PROGRAM MAIN
VAR
	// ------ Linking variables to IO cards ------
		// --------- Outputs ---------
	Flow_Valve_1 	AT %Q* : INT;
	Level_Valve_1 	AT %Q* : INT;
	Level_Valve_2 	AT %Q* : INT;
	Level_Valve_3 	AT %Q* : INT;
	Gas_Valve 		AT %Q* : INT;
	Mixer_Valve 	AT %Q* : INT;
	Motor_speed 	AT %Q* : INT;	
	Motor_Direction AT %Q* : BOOL; 			// Don't touch
		// --------- Inputs ---------
			// Buttons
	Toggle_Button 	AT %I* :BOOL;	// Normally Open  (OFF), Green
	Reset_Button 	AT %I* : BOOL; 	// Normally Closed (ON), Red
	EMERGENCY_STOP 	AT %I* : BOOL; 	// Normally Closed (ON), Emergency Switch
			// Sensors
	Level_Transmitter_1 	AT %I* :INT;
	Level_Transmitter_2 	AT %I* :INT;
	Temperature_Transmitter AT %I* :INT;
	Pressure_Differencial_Transmitter_1 AT %I* : INT;
	Pressure_Differencial_Transmitter_2 AT %I* : INT;
	Pressure_Transmitter_1 AT %I* : INT ;
	Pressure_Transmitter_2 AT %I* : INT ;
	Pressure_Transmitter_3 AT %I* : INT ; 
	// ------ Linking variables to IO cards ------
	
	// ------- Display Input Variables ---------
		// Percentages
	LT1percent  : INT;
	LT2percent  : INT;
	TT1percent  : INT;
	PDT1percent : INT;
	PDT2percent : INT;
	PT1percent  : INT;
	PT2percent  : INT;
	PT3percent  : INT;
		// Actual values
	LT1mm 	: REAL;
	LT2mm 	: REAL;
	TT1c 	: REAL;
	PDT1bar : REAL;
	PDT2bar : REAL;
	PT1bar  : REAL;
	PT2bar  : REAL;
	PT3bar  : REAL;
		// Scaling variables
	bitMax 		: REAL := 32767;			// [bits]
	minPT 		: REAL := 0.06;				// [bar]
	maxPT 		: REAL := 6;				// [bar]
	deltaPT 	: REAL := maxPT - minPT;	// [bar]
	minPDT		: REAL := 0.004;			// [bar]
	maxPDT		: REAL := 0.4;				// [bar]
	deltaPDT	: REAL := maxPDT - minPDT;	// [bar]
	
	//maxLT 		: REAL := 304.8;			// [mm]
	minLT1  	: REAL := 37.0;				// [mm]
	minLT1bit  	: REAL := 270.0;			// [mm]
	minLT2  	: REAL := 42.0;				// [mm]
	kLT1		: REAL := 9.0/1694.0;		// [deltaMMmeasured/deltaBitmeasured]
	kLT2		: REAL := 9.0/1529.0;		// [deltaMMmeasured/deltaBitmeasured
	
	maxTT		: REAL := 250;				// [celsius]
	minTT		: REAL := -50;				// [celsius]
	deltaTT 	: REAL := maxTT - minTT;	// [celsius]
	// ------- Display Input Variables --------- 
	
	
		// Toggle Motor Statee with green button
	risingEdge : R_TRIG;
	elapsedDebounce : TIME;
	toggleMotor : BOOL;
	
	// ------------------ HMI ------------------
	Motor_ON : BOOL; 				// For HMI button
	ON_OFF 	 : STRING(10) := 'OFF'; // For HMI text
	// ------------------ HMI ------------------
	
	// Emergency System
	alarmSystem : FB_AlarmSystem;
	
	// Initializer
	init : BOOL := FALSE;
	mainInitializer : FB_defaultValues;
END_VAR

VAR_INPUT
	Motor_ON_OFF 	AT %Q* : BOOL := FALSE;	// Motor switch	
	// User Input as percentage, Declaration
	Flow_Valve_1_Percentage	: INT;	// Start values
	Level_Valve_1_Percentage: INT;	// From Manual
	Level_Valve_2_Percentage: INT;
	Level_Valve_3_Percentage: INT;
	Motor_speed_Percentage	: INT; // Start speed, ideal: 30-35%
END_VAR


// ======================== Initializer ========================
	IF NOT init THEN
		mainInitializer(MotorState  := Motor_ON_OFF,
						MotorSpeed  := Motor_speed_Percentage,
						FV1_Percent := Flow_Valve_1_Percentage,
						LV1_Percent := Level_Valve_1_Percentage,
						LV2_Percent := Level_Valve_2_Percentage,
						LV3_Percent := Level_Valve_3_Percentage);
		init := TRUE;
	END_IF
// ======================== Initializer ========================

// ======================== Alarm System ========================
	alarmSystem(ClearButton := Reset_Button,
				EmergencyButton := EMERGENCY_STOP);
// ======================== Alarm System ========================
	
// ================ Outer bounds logic (outputs) ================
IF Flow_Valve_1_Percentage > 100 THEN
	Flow_Valve_1_Percentage := 100; 
	ELSE IF Flow_Valve_1_Percentage < 0 THEN 
		Flow_Valve_1_Percentage := 0; 
	END_IF
END_IF

IF Level_Valve_1_Percentage > 100 THEN
	Level_Valve_1_Percentage := 100; 
	ELSE IF Level_Valve_1_Percentage < 0 THEN 
		Level_Valve_1_Percentage := 0; 
	END_IF
END_IF

IF Level_Valve_2_Percentage > 100 THEN
	Level_Valve_2_Percentage := 100; 
	ELSE IF Level_Valve_2_Percentage < 0 THEN 
		Level_Valve_2_Percentage := 0; 
	END_IF
END_IF

IF Level_Valve_3_Percentage > 100 THEN
	Level_Valve_3_Percentage := 100; 
	ELSE IF Level_Valve_3_Percentage < 0 THEN 
		Level_Valve_3_Percentage := 0; 
	END_IF
END_IF

IF Motor_speed_Percentage > 100 THEN
	Motor_speed_Percentage := 100; 
	ELSE IF Motor_speed_Percentage < 0 THEN 
		Motor_speed_Percentage := 0; 
	END_IF
END_IF
// ================= Outer bounds logic (outputs) ================

// ================= Percentage Mapping (OUTPUTS) =================
	// Take 2 [V] to 10 [V]
// Flow_Valve_1 calibration
Flow_Valve_1 := REAL_TO_INT (262.14*Flow_Valve_1_Percentage +6553 ); 
// Level_Valve_1 calibration
Level_Valve_1 := REAL_TO_INT(262.14*Level_Valve_1_Percentage +6553);
// Level_Valve_2 calibration
Level_Valve_2 := REAL_TO_INT(262.14*Level_Valve_2_Percentage +6553);
// Level_Valve_3 calibration
Level_Valve_3 := REAL_TO_INT(262.14*Level_Valve_3_Percentage +6553);

// Motor_speed calibration
Motor_speed := REAL_TO_INT(262.14*Motor_speed_Percentage +6553);
// ================= Percentage Mapping (OUTPUTS) =================

// ================= Mapping (INPUTS) =================
		// Take 4 [mA] to 20 [mA] 
	// Percentages
	LT1percent  := Level_Transmitter_1;
	LT2percent  := Level_Transmitter_2;
	TT1percent  := Temperature_Transmitter;
	PDT1percent := Pressure_Differencial_Transmitter_1;
	PDT2percent := Pressure_Differencial_Transmitter_2;
	PT1percent  := Pressure_Transmitter_1;
	PT2percent  := Pressure_Transmitter_2;
	PT3percent  := Pressure_Transmitter_3;
		// Actual values
	LT1mm 	:= Level_Transmitter_1					* kLT1 						+ minLT1; // Different Mapping
	LT2mm 	:= Level_Transmitter_2 					* kLT2						+ minLT2; // Different Mapping
	TT1c 	:= Temperature_Transmitter 				* (deltaTT/bitMax)  		+ minTT;
	PDT1bar := Pressure_Differencial_Transmitter_1 	* (deltaPDT/bitMax) 		+ minPDT;
	PDT2bar := Pressure_Differencial_Transmitter_2 	* (deltaPDT/bitMax) 		+ minPDT;
	PT1bar  := Pressure_Transmitter_1 				* (deltaPT/bitMax)  		+ minPT;
	PT2bar  := Pressure_Transmitter_2 				* (deltaPT/bitMax)  		+ minPT;
	PT3bar  := Pressure_Transmitter_3 				* (deltaPT/bitMax)  		+ minPT;

	(*IF (LT1mm < 40.0) THEN
		LT1mm := 0.0;
	END_IF
	IF (LT2mm < 0.0) THEN
		LT2mm := 0.0;
	END_IF*)
// ================= Mapping (INPUTS) =================

	// Toggle motor state with green button
risingEdge(CLK := Toggle_Button,
		   Q => toggleMotor);
IF toggleMotor THEN
	Motor_ON_OFF := NOT Motor_ON_OFF;
END_IF

// ======================== HMI Display ========================
 // Start motor?
IF Motor_ON_OFF   THEN
    Motor_ON   :=  FALSE;		// Button display
	ON_OFF  := 'MOTOR: ON' ;	// Text display
	
ELSE
    Motor_ON  := TRUE;			// Button display
	ON_OFF  := 'MOTOR: OFF' ;	// Text display
END_IF
// ======================== HMI Display ========================

END_PROGRAM

(* stored: Version 1.1.0.1, ProductVersion 3.1.4024.12
   POU MAIN: Id {75317203-8f43-4932-aa88-c7b05e9ca563}, SpecialFunc None *)
